(* PLC project Unnamed, Unknown Unnamed 1 *)
(* stored: creationDateTime 2026-01-20T18:46:13, modificationDateTime 2026-01-20T18:46:13 *)

PROGRAM main
  VAR
    PB1 AT %IX0.0 : BOOL;
    LED1 AT %QX0.0 : BOOL;
  END_VAR
  VAR
    Blink_Status : BOOL;
    Blink_Timer1 : TON;
    Blink_Timer2 : TOF;
    Wait_Time : TIME := T#2s;
    TON0 : TON;
    TOF0 : TOF;
  END_VAR

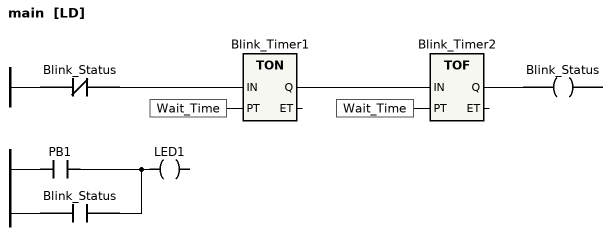
(* LD diagram, written out as Structured Text *)
Blink_Timer1(IN := NOT Blink_Status, PT := Wait_Time);
Blink_Timer2(IN := Blink_Timer1.Q, PT := Wait_Time);
Blink_Status := Blink_Timer2.Q;
LED1 := PB1 OR Blink_Status;
END_PROGRAM

CONFIGURATION Config0
  RESOURCE Res0 ON PLC
    TASK task0(INTERVAL := T#20ms, PRIORITY := 1);
    PROGRAM instance0 WITH task0 : main;
  END_RESOURCE
END_CONFIGURATION
